FUNCTION Convert_TIME_TO_INT : BOOL
VAR_INPUT
	in : TIME;
	out : REFERENCE TO INT;
END_VAR
VAR
	converted : INT;
END_VAR

converted := TIME_TO_INT(in);

IF (INT_TO_TIME(converted) <> in) THEN
	RETURN;
END_IF

out := converted;
Convert_TIME_TO_INT := TRUE;

END_FUNCTION

(* stored: Version 1.1.0.1, ProductVersion 3.1.4024.12
   POU Convert_TIME_TO_INT: Id {94920137-97b2-4853-868b-398f8a0e0f70}, SpecialFunc None *)
